// TIA Portal V19 export
TYPE "LUC_typeModeConfiguration"
TITLE = LUC_typeModeConfiguration
// Configure which modes are enabled
// stored: Access Published
   STRUCT
      production : Bool := true;   // Enable unit mode Production
      maintenance : Bool := true;   // Enable unit mode Maintenance
      manual : Bool := true;   // Enable mode Manual (Mandatory, always set)
      userMode01 : Bool;   // Enable user-defined unit mode 01
      userMode02 : Bool;   // Enable user-defined unit mode 02
      userMode03 : Bool;   // Enable user-defined unit mode 03
      userMode04 : Bool;   // Enable user-defined unit mode 04
      userMode05 : Bool;   // Enable user-defined unit mode 05
      userMode06 : Bool;   // Enable user-defined unit mode 06
      userMode07 : Bool;   // Enable user-defined unit mode 07
      userMode08 : Bool;   // Enable user-defined unit mode 08
      userMode09 : Bool;   // Enable user-defined unit mode 09
      userMode10 : Bool;   // Enable user-defined unit mode 10
      userMode11 : Bool;   // Enable user-defined unit mode 11
      userMode12 : Bool;   // Enable user-defined unit mode 12
      userMode13 : Bool;   // Enable user-defined unit mode 13
   END_STRUCT;
END_TYPE
